{attribute 'GeneratedUsingTerminal: EP7041-0002-0016'}
{attribute addProperty BoxType "EP7041-0002-0016"}
{attribute addProperty Id "StatusAT %I*Status_8CBE219F12Counter_valueAT %I*UINT2Latch_valueAT %I*UINT2"}
{attribute addProperty CRC "1292267034"}
{attribute addProperty Size "16"}
TYPE ENC_Status_compact_4D066E1A :
STRUCT
	{attribute addProperty Name "Status"}
	Status AT %I* : Status_8CBE219F;
	{attribute addProperty Name "Counter_value"}
	Counter_value AT %I* : UINT;
	{attribute addProperty Name "Latch_value"}
	Latch_value AT %I* : UINT;
END_STRUCT
END_TYPE

(* stored: Version 1.2.0.0, ProductVersion 3.1.4024.9
   DUT ENC_Status_compact_4D066E1A: Id {fadf6159-ad54-40d0-9232-08d5ff8c4416} *)
